(* CODESYS project Studienarbeits_Projekt.project

Project tree, tasks and I/O mapping:
  Device : CODESYS SoftMotion Win V3, 3S - Smart Software Solutions GmbH, version 3.5.18.30
    application Application
      libraries: SysTypes Interfaces, * (System); SysFile, 3.5.17.0 (System); Standard, 3.5.18.0 (System)
      task Scara_PlanningTask (cyclic, interval t#8ms, priority 2) calls Scara_PlanningPrg
      task Achsen (cyclic, interval T#3ms, priority 1) calls Roboter, Fertigung, NC4
      visualisation VIS_Arm2
      program Scara_PlanningPrg [ST]
      global variables GVL
      axis group Scara: TRAFO.Kin_Scara2_Z, axes Motor1, Motor2, Motor3
      trace Sampling_Trace (task ): 
      program Roboter [FBD]
      function Dist [ST]
      visualisation Fertigungszelle
      program Fertigung [SFC]: Ziel2, Ziel3, Ziel1
      visualisation VIS_Arm2_1
      program NC4 [FBD]
      visualisation InputImage
      visualisation OutputImage
    SoftMotion General Axis Pool
      Motor4 : SM_Drive_Virtual, 3S - Smart Software Solutions GmbH, order no. 1805, version 4.0.0.0
          settings: wDriveID = 2; fSWMaxVelocity = 1e3; fSWMaxAcceleration = 1e5; fSWMaxDeceleration = 1e5; fRampJerk = 1e7
      Motor1 : SM_Drive_Virtual, 3S - Smart Software Solutions GmbH, order no. 1805, version 4.0.0.0
          settings: fSWMaxVelocity = 1e3; fSWMaxAcceleration = 1e5; fSWMaxDeceleration = 1e5; fRampJerk = 1e7; fSWLimitPositive = 180; fSWLimitNegative = -180
      Motor2 : SM_Drive_Virtual, 3S - Smart Software Solutions GmbH, order no. 1805, version 4.0.0.0
          settings: fSWMaxVelocity = 1e3; fSWMaxAcceleration = 1e5; fSWMaxDeceleration = 1e5; fRampJerk = 1e7; fSWLimitPositive = 180; fSWLimitNegative = -180
      Motor3 : SM_Drive_Virtual, 3S - Smart Software Solutions GmbH, order no. 1805, version 4.0.0.0
          settings: wDriveID = 3; fSWMaxVelocity = 1e3; fSWMaxAcceleration = 1e5; fSWMaxDeceleration = 1e5; fRampJerk = 1e7; fSWLimitPositive = 110.0
  libraries: VisuSymbols, 4.1.0.0 (System); SM3_Basic, 4.12.0.0 (3S - Smart Software Solutions GmbH)
  text list GlobalTextList
  GlobalImagePool
*)

// Device/Application/GVL
VAR_GLOBAL
	NotAus: BOOL;
	p_Ziel, p_Ist: SMC_POS_REF;
	PTPMove: BOOL;
	LinMove: BOOL;
	AxisMove: BOOL;
	Start: BOOL;
	Objekt_erkannt: BOOL;
	p_Band:MC_COORD_REF:=(x:=-146,y:=106,z:=0,a:=0,b:=0,c:=0);
	p_init:MC_COORD_REF:=(x:=27,y:=-11,z:=0,a:=0,b:=0,c:=0);
	Zugreifen: BOOL;
	Schrauben: BOOL;
	CoordSystem: SMC_COORD_SYSTEM;
	p_Start: SMC_POS_REF;
	StopTracking: BOOL;
	StartTracking: BOOL;
	Stop: BOOL;
	//Bildverarbeitung
	pic_width	 : INT := 48; 	(* Bildbreite in Pixel *)
	X			: INT;			(* X-Position Merkmal *)
	Y 			: INT;	 		(* Y-Position Merkmal *)
	BV_Start: BOOL;
	BV_Fertig: BOOL;
END_VAR
VAR_GLOBAL CONSTANT
	PI: REAL := 3.141592654;
END_VAR

// Device/Application/Scara_PlanningPrg
PROGRAM Scara_PlanningPrg

;

END_PROGRAM

// Device/Application/Roboter
PROGRAM Roboter
VAR
	GroupEnable: MC_GroupEnable;
	MoveDirectAbsolute: MC_MoveDirectAbsolute;
	MoveLinearAbsolute: MC_MoveLinearAbsolute;
	E1,E2,E3:MC_Power;
	TCP:MC_GroupReadActualPosition;
	Axes: MC_GroupReadActualPosition;
	NC3: MC_MoveAbsolute;
END_VAR

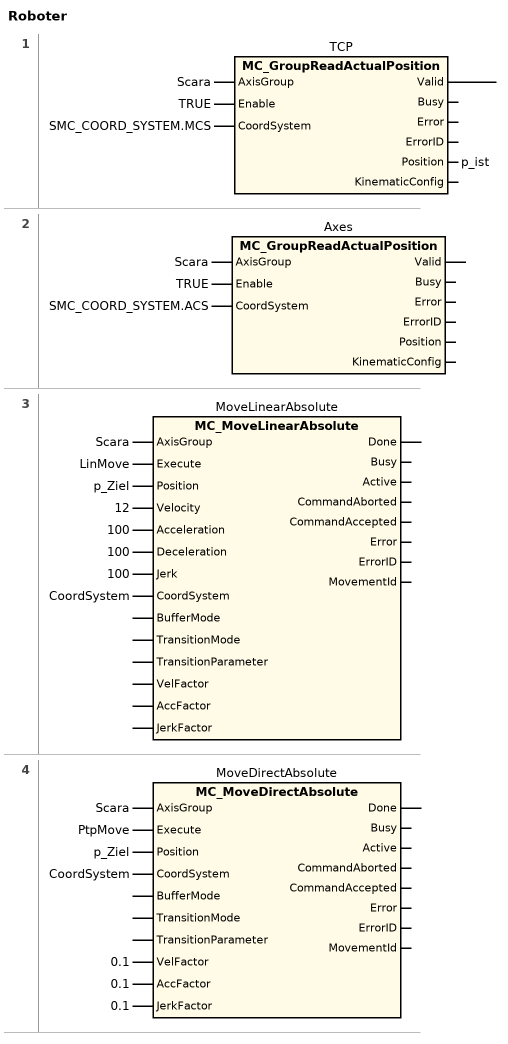
// NETWORK 1
TCP(AxisGroup := Scara, Enable := TRUE, CoordSystem := SMC_COORD_SYSTEM.MCS, Position => p_ist); // MC_GroupReadActualPosition

// NETWORK 2
Axes(AxisGroup := Scara, Enable := TRUE, CoordSystem := SMC_COORD_SYSTEM.ACS); // MC_GroupReadActualPosition

// NETWORK 3
MoveLinearAbsolute(
    AxisGroup := Scara,
    Execute := LinMove,
    Position := p_Ziel,
    Velocity := 12,
    Acceleration := 100,
    Deceleration := 100,
    Jerk := 100,
    CoordSystem := CoordSystem); // MC_MoveLinearAbsolute

// NETWORK 4
MoveDirectAbsolute(
    AxisGroup := Scara,
    Execute := PtpMove,
    Position := p_Ziel,
    CoordSystem := CoordSystem,
    VelFactor := 0.1,
    AccFactor := 0.1,
    JerkFactor := 0.1); // MC_MoveDirectAbsolute

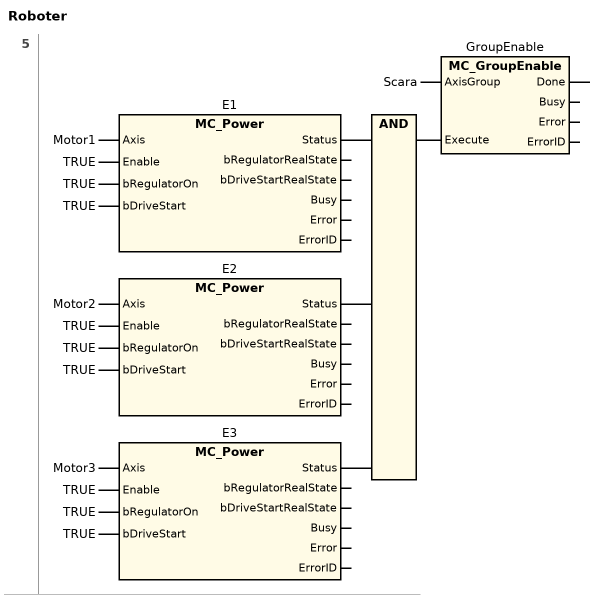
// NETWORK 5
E1(Axis := Motor1, Enable := TRUE, bRegulatorOn := TRUE, bDriveStart := TRUE); // MC_Power
E2(Axis := Motor2, Enable := TRUE, bRegulatorOn := TRUE, bDriveStart := TRUE); // MC_Power
E3(Axis := Motor3, Enable := TRUE, bRegulatorOn := TRUE, bDriveStart := TRUE); // MC_Power
GroupEnable(AxisGroup := Scara, Execute := E1.Status AND E2.Status AND E3.Status); // MC_GroupEnable

END_PROGRAM

// Device/Application/Fertigung
PROGRAM Fertigung
VAR
	SFCCurrentStep:STRING;
	b:ARRAY[1..2] OF INT:=[36,7];
	c:ARRAY[1..3] OF REAL:=[-74,-38,100];
	u_M:INT:=24;
	v_M:INT:=18;
	lambda_v:REAL:=0.1; (* mm/PIXel *)
	lambda_u:REAL:=0.1; (* mm/PIXel *)
	f: REAL:=10; (* mm Brennweite *)
END_VAR

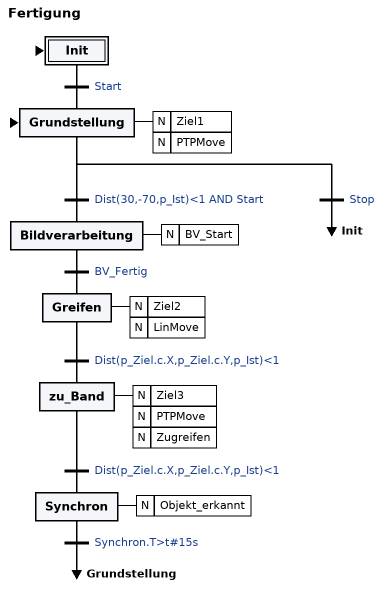
INITIAL_STEP Init:
END_STEP
TRANSITION FROM Init TO Grundstellung
    := Start;
END_TRANSITION
STEP Grundstellung:
    Ziel1(N);
    PTPMove(N);
END_STEP
TRANSITION FROM Grundstellung TO Bildverarbeitung
    := Dist(30,-70,p_Ist)<1 AND Start;
END_TRANSITION
TRANSITION FROM Grundstellung TO Init
    := Stop;
END_TRANSITION
STEP Bildverarbeitung:
    BV_Start(N);
END_STEP
TRANSITION FROM Bildverarbeitung TO Greifen
    := BV_Fertig;
END_TRANSITION
STEP Greifen:  // min time t#5s
    Ziel2(N);
    LinMove(N);
END_STEP
TRANSITION FROM Greifen TO zu_Band
    := Dist(p_Ziel.c.X,p_Ziel.c.Y,p_Ist)<1;
END_TRANSITION
STEP zu_Band:  // min time t#5s
    Ziel3(N);
    PTPMove(N);
    Zugreifen(N);
END_STEP
TRANSITION FROM zu_Band TO Synchron
    := Dist(p_Ziel.c.X,p_Ziel.c.Y,p_Ist)<1;
END_TRANSITION
STEP Synchron:
    Objekt_erkannt(N);
END_STEP
TRANSITION FROM Synchron TO Grundstellung
    := Synchron.T>t#15s;
END_TRANSITION

ACTION Ziel2:
CoordSystem:=SMC_Coord_System.MCS;
p_ZIEL.c.x:=-85;
p_ZIEL.c.y:=-50;
p_ZIEL.c.z:=0;
END_ACTION

ACTION Ziel3:
CoordSystem:=SMC_Coord_System.MCS;
p_Ziel.c.x:=-100;
p_Ziel.c.y:=80;
p_Ziel.c.z:=0;
END_ACTION

ACTION Ziel1:
CoordSystem:=SMC_Coord_System.MCS;
p_ZIEL.c.X:=30;
p_ZIEL.c.Y:=-70;
p_ZIEL.c.Z:=0;
END_ACTION

END_PROGRAM

// Device/Application/NC4
 PROGRAM NC4
VAR
	E4:MC_Power;
	N4: MC_MoveVelocity;
	Reset: MC_SetPosition;
	Event: R_TRIG;
	Objekt: RS;
END_VAR

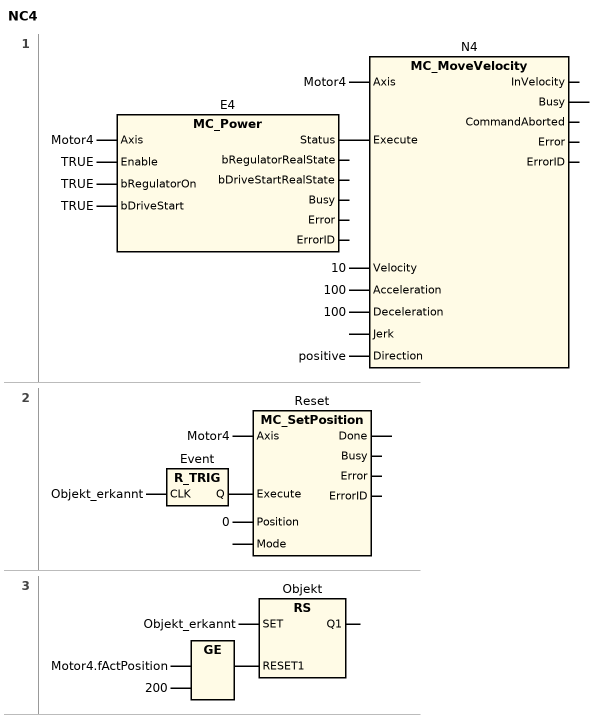
// NETWORK 1
E4(Axis := Motor4, Enable := TRUE, bRegulatorOn := TRUE, bDriveStart := TRUE); // MC_Power
N4(
    Axis := Motor4,
    Execute := E4.Status,
    Velocity := 10,
    Acceleration := 100,
    Deceleration := 100,
    Direction := positive); // MC_MoveVelocity

// NETWORK 2
Event(CLK := Objekt_erkannt); // R_TRIG
Reset(Axis := Motor4, Execute := Event.Q, Position := 0); // MC_SetPosition

// NETWORK 3
Objekt(SET := Objekt_erkannt, RESET1 := Motor4.fActPosition >= 200); // RS

END_PROGRAM

// Device/Application/Dist
FUNCTION Dist : LREAL
VAR_INPUT
	x_Soll, y_Soll:  LREAL;
	p_Ist: SMC_POS_REF;
END_VAR
VAR
END_VAR

Dist:=SQRT((x_SOLL-p_IST.c.X)*(x_SOLL-p_IST.c.X)+(y_SOLL-p_IST.c.Y)*(y_SOLL-p_IST.c.Y));

END_FUNCTION

// Device/Application/VIS_Arm2
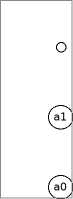
VISUALIZATION VIS_Arm2  // 73x199
VAR_IN_OUT(*	qAct:ARRAY[1..6] OF REAL;*)
	qAct:TRAFO.AXISPOS_REF;
	pAct:MC_COORD_REF;
	Tool:BOOL;
END_VAR
    Polygon (65,105)
        p3560616238: 70*COS(qAct.a0*PI/180)
        p2738717112: 70*(1-SIN(qAct.a0*PI/180))
        p2858320360: 90-(qAct.a1+qAct.a0)
    Polygon (65,175)
        p2858320360: 90-qAct.a0
    Ellipse (48,175 25x24), "a0"
    Ellipse (48,105 25x24), "a1"
        p3560616238: 70*COS(qAct.a0*PI/180)
        p2738717112: 70*(1-SIN(qAct.a0*PI/180))
    Ellipse (56,42 10x10), colour toggle: Tool
        p3560616238: pAct.X
        p2738717112: 140-pAct.Y
END_VISUALIZATION

// Device/Application/Fertigungszelle
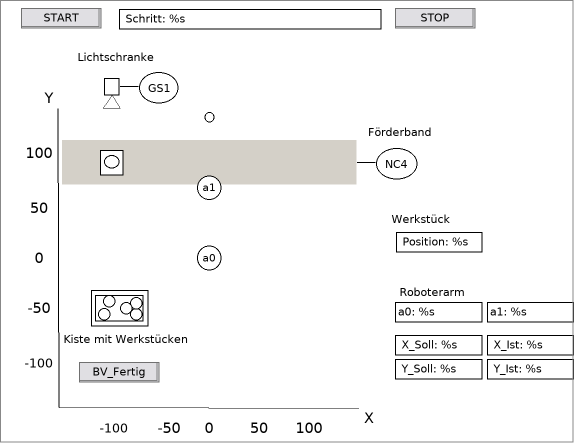
VISUALIZATION Fertigungszelle  // 574x443
    Ellipse (376,148 41x31), colour toggle: NC4.N4.Busy
    RoundedRectangle (62,140 294x44)
    Rectangle (91,290 57x36)
    Rectangle (95,295 48x26)
    Ellipse (98,308 12x12)
    Ellipse (130,308 12x12), colour toggle: Zugreifen
    Ellipse (130,297 12x12), colour toggle: Zugreifen
    Ellipse (120,302 12x12), colour toggle: Zugreifen
    Ellipse (103,295 12x12), colour toggle: Zugreifen
    Rectangle (57,321 138x37), "Kiste mit Werkstücken"
    Polyline (195,85)
    Line (59,407) (58,108)
    Line (59,407) (358,408)
    Polyline (345,235)
    Rectangle (359,408 20x20), "X"
    Rectangle (39,88 20x20), "Y"
    Rectangle (24,243 30x30), "0"
    Rectangle (194,413 30x30), "0"
    Rectangle (244,413 30x30), "50"
    Rectangle (154,413 30x30), "-50"
    Rectangle (294,413 30x30), "100"
    Rectangle (99,413 30x30), "-100"
    Rectangle (24,193 30x30), "50"
    Rectangle (24,138 30x30), "100"
    Rectangle (24,293 30x30), "-50"
    Rectangle (24,348 30x30), "-100"
    Button (21,8 80x20), "START"
        tap START
    Rectangle (119,9 262x20), "Schritt: %s", text variable: Fertigung.SFCCurrentStep
    Rectangle (100,150 23x25), invisible if: NOT NC4.Objekt.Q1
        p3560616238: Motor4.fActPosition
    Ellipse (104,155 15x13), invisible if: NOT NC4.Objekt.Q1
        p3560616238: Motor4.fActPosition
    Rectangle (104,78 15x17)
    Polygon (103,108) (120,108) (112,95)
    Frame (152,70 69x200)
        shows VIS_Arm2(qAct := Roboter.Axes.Position.a, pAct := Roboter.TCP.Position.c, Tool := Schrauben OR Zugreifen)
    Button (79,362 80x20), "BV_Fertig"
        tap BV_Fertig
    Rectangle (395,335 87x20), "X_Soll: %s", text variable: p_ZIEL.c.X
    Rectangle (487,335 87x20), "X_Ist: %s", text variable: p_Ist.c.X
    Rectangle (395,359 87x20), "Y_Soll: %s", text variable: p_ZIEL.c.Y
    Rectangle (487,359 87x20), "Y_Ist: %s", text variable: p_Ist.c.Y
    Rectangle (62,39 108x37), "Lichtschranke"
    Rectangle (395,302 87x20), "a0: %s", text variable: Roboter.Axes.Position.a.a0
    Rectangle (487,302 87x20), "a1: %s", text variable: Roboter.Axes.Position.a.a1
    Rectangle (396,232 86x20), "Position: %s", text variable: Motor4.fActPosition, invisible if: Not NC4.Objekt.Q1
    Rectangle (378,274 108x37), "Roboterarm"
    Rectangle (367,201 108x37), "Werkstück", invisible if: Not NC4.Objekt.Q1
    Rectangle (381,149 31x31), "NC4"
    Rectangle (346,114 108x37), "Förderband"
    Line (357,162)
    Line (356,162)
    Line (357,162) (375,162)
    Ellipse (139,72 39x31), colour toggle: Objekt_erkannt
    Rectangle (144,73 31x31), "GS1", colour toggle: Objekt_erkannt
    Line (120,86)
    Line (119,86)
    Line (120,86) (138,86)
    Button (395,8 80x20), "STOP"
        tap Stop
END_VISUALIZATION

// Device/Application/VIS_Arm2_1
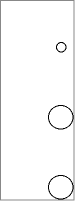
VISUALIZATION VIS_Arm2_1  // 75x201
VAR_IN_OUT(*	qAct:ARRAY[1..6] OF REAL;*)
	qAct:TRAFO.AXISPOS_REF;
	pAct:MC_COORD_REF;
END_VAR
    Polygon (65,105)
        p3560616238: 70*COS(qAct.a0*PI/180)
        p2738717112: 70*(1-SIN(qAct.a0*PI/180))
        p2858320360: 90-(qAct.a1+qAct.a0)
    Polygon (65,175)
        p2858320360: 90-qAct.a0
    Ellipse (48,175 25x24)
    Ellipse (48,105 25x24)
        p3560616238: 70*COS(qAct.a0*PI/180)
        p2738717112: 70*(1-SIN(qAct.a0*PI/180))
    Ellipse (56,42 10x10), colour toggle: pAct.Z>1
        p3560616238: pAct.X
        p2738717112: 140-pAct.Y
END_VISUALIZATION

// Device/Application/InputImage
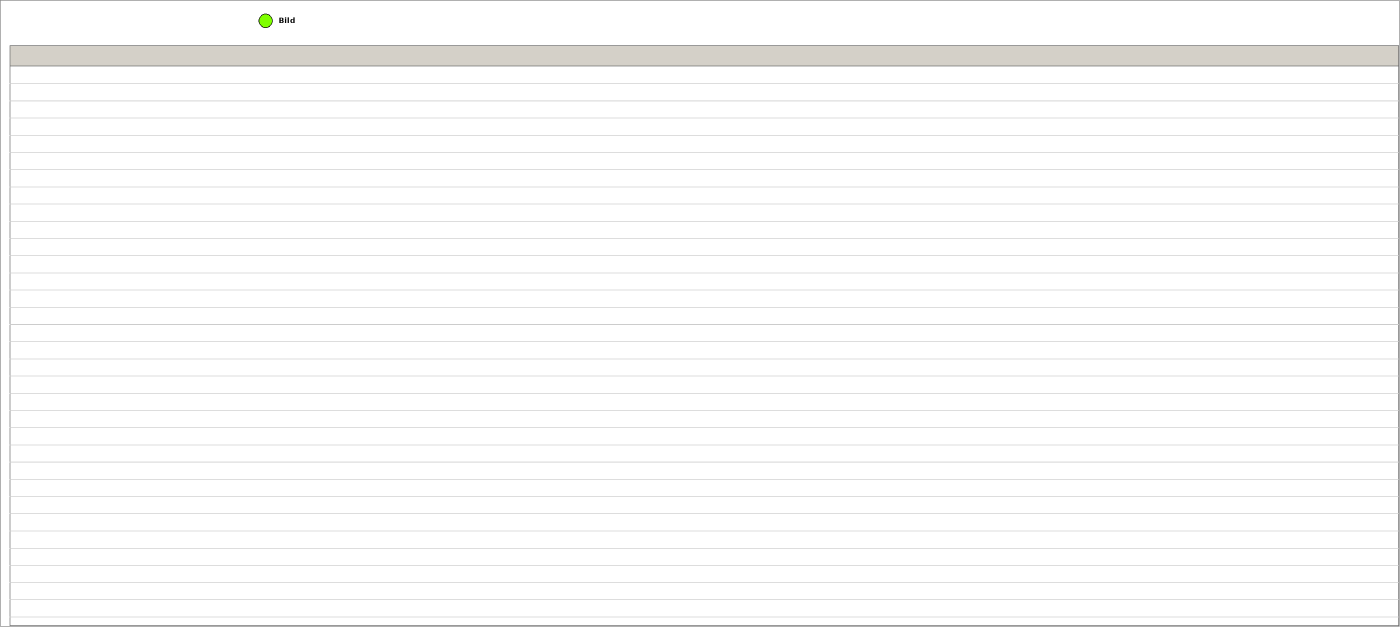
VISUALIZATION InputImage  // 2031x911
    Ellipse (375,20 20x20), colour toggle: BV_Start
        tap BV_Start
    Rectangle (401,20 32x20), "Bild"
    Table (14,66 2015x843), data array: BV.PicArray
        p3854506369: BV.PicArray[0,INDEX]
        p1892666644: BV.PicArray[1,INDEX]
        p338671338: BV.PicArray[2,INDEX]
        p2170511999: BV.PicArray[3,INDEX]
        p3723444502: BV.PicArray[4,INDEX]
        p1218418051: BV.PicArray[5,INDEX]
        p746581629: BV.PicArray[6,INDEX]
        p3104783080: BV.PicArray[7,INDEX]
        p2501879983: BV.PicArray[8,INDEX]
        p7306298: BV.PicArray[9,INDEX]
        p1933151965: BV.PicArray[10,INDEX]
        p3863566920: BV.PicArray[11,INDEX]
        p2192122294: BV.PicArray[12,INDEX]
        p400160035: BV.PicArray[13,INDEX]
        p1265227338: BV.PicArray[14,INDEX]
        p3726181087: BV.PicArray[15,INDEX]
        p3136911649: BV.PicArray[16,INDEX]
        p797552052: BV.PicArray[17,INDEX]
        p60375027: BV.PicArray[18,INDEX]
        p2531912550: BV.PicArray[19,INDEX]
        p693678525: BV.PicArray[20,INDEX]
        p3156763944: BV.PicArray[21,INDEX]
        p3636993750: BV.PicArray[22,INDEX]
        p1303956035: BV.PicArray[23,INDEX]
        p285796650: BV.PicArray[24,INDEX]
        p2222472639: BV.PicArray[25,INDEX]
        p3768075841: BV.PicArray[26,INDEX]
        p1978176212: BV.PicArray[27,INDEX]
        p1509425299: BV.PicArray[28,INDEX]
        p3431519238: BV.PicArray[29,INDEX]
        p2846402210: BV.PicArray[30,INDEX]
        p1020817975: BV.PicArray[31,INDEX]
        p1480067529: BV.PicArray[32,INDEX]
        p3444104540: BV.PicArray[33,INDEX]
        p2449014325: BV.PicArray[34,INDEX]
        p76032672: BV.PicArray[35,INDEX]
        p1617449310: BV.PicArray[36,INDEX]
        p4112025035: BV.PicArray[37,INDEX]
        p3641186188: BV.PicArray[38,INDEX]
        p1282982681: BV.PicArray[39,INDEX]
        p2644168573: BV.PicArray[40,INDEX]
        p149560296: BV.PicArray[41,INDEX]
        p1812619286: BV.PicArray[42,INDEX]
        p4185568387: BV.PicArray[43,INDEX]
        p2781517802: BV.PicArray[44,INDEX]
        p817513343: BV.PicArray[45,INDEX]
        p1415198849: BV.PicArray[46,INDEX]
        p3240815636: BV.PicArray[47,INDEX]
        p3980033619: BV.PicArray[48,INDEX]
END_VISUALIZATION

// Device/Application/OutputImage
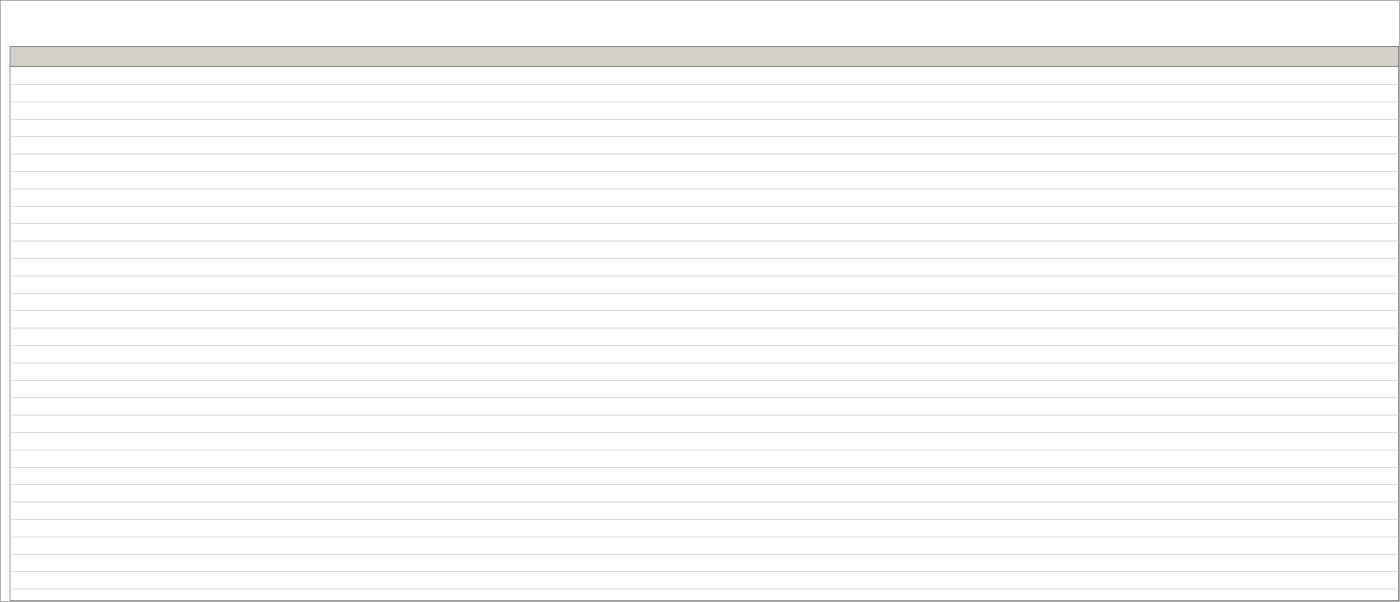
VISUALIZATION OutputImage  // 2009x865
    Table (14,66 1993x797), data array: BV.ObjArray
        p3854506369: BV.ObjArray[0,INDEX]
        p1892666644: BV.ObjArray[1,INDEX]
        p338671338: BV.ObjArray[2,INDEX]
        p2170511999: BV.ObjArray[3,INDEX]
        p3723444502: BV.ObjArray[4,INDEX]
        p1218418051: BV.ObjArray[5,INDEX]
        p746581629: BV.ObjArray[6,INDEX]
        p3104783080: BV.ObjArray[7,INDEX]
        p2501879983: BV.ObjArray[8,INDEX]
        p7306298: BV.ObjArray[9,INDEX]
        p1933151965: BV.ObjArray[10,INDEX]
        p3863566920: BV.ObjArray[11,INDEX]
        p2192122294: BV.ObjArray[12,INDEX]
        p400160035: BV.ObjArray[13,INDEX]
        p1265227338: BV.ObjArray[14,INDEX]
        p3726181087: BV.ObjArray[15,INDEX]
        p3136911649: BV.ObjArray[16,INDEX]
        p797552052: BV.ObjArray[17,INDEX]
        p60375027: BV.ObjArray[18,INDEX]
        p2531912550: BV.ObjArray[19,INDEX]
        p693678525: BV.ObjArray[20,INDEX]
        p3156763944: BV.ObjArray[21,INDEX]
        p3636993750: BV.ObjArray[22,INDEX]
        p1303956035: BV.ObjArray[23,INDEX]
        p285796650: BV.ObjArray[24,INDEX]
        p2222472639: BV.ObjArray[25,INDEX]
        p3768075841: BV.ObjArray[26,INDEX]
        p1978176212: BV.ObjArray[27,INDEX]
        p1509425299: BV.ObjArray[28,INDEX]
        p3431519238: BV.ObjArray[29,INDEX]
        p2846402210: BV.ObjArray[30,INDEX]
        p1020817975: BV.ObjArray[31,INDEX]
        p1480067529: BV.ObjArray[32,INDEX]
        p3444104540: BV.ObjArray[33,INDEX]
        p2449014325: BV.ObjArray[34,INDEX]
        p76032672: BV.ObjArray[35,INDEX]
        p1617449310: BV.ObjArray[36,INDEX]
        p4112025035: BV.ObjArray[37,INDEX]
        p3641186188: BV.ObjArray[38,INDEX]
        p1282982681: BV.ObjArray[39,INDEX]
        p2644168573: BV.ObjArray[40,INDEX]
        p149560296: BV.ObjArray[41,INDEX]
        p1812619286: BV.ObjArray[42,INDEX]
        p4185568387: BV.ObjArray[43,INDEX]
        p2781517802: BV.ObjArray[44,INDEX]
        p817513343: BV.ObjArray[45,INDEX]
        p1415198849: BV.ObjArray[46,INDEX]
        p3240815636: BV.ObjArray[47,INDEX]
        p3980033619: BV.ObjArray[48,INDEX]
END_VISUALIZATION
